(* PLC project liner_cyclic.project, CODESYS CODESYS V3.5 SP17 Patch 3 *)
(* stored: creationDateTime 1970-01-01T00:00:00, modificationDateTime 1970-01-01T00:00:00 *)

FUNCTION StartAfterReadingInputs : DWORD
  VAR_IN_OUT
    EventPrm : CmpIecTask.EVTPARAM_CmpIecTask;
  END_VAR

            //GVL.bMainDelay := TRUE;
          
END_FUNCTION
